PROGRAM MAIN
VAR
	
axis: AXIS_REF;
power: MC_POWER();

limNeg AT %I* :BOOL;
limPos AT %I*:BOOL;


EPSlimNeg AT %I* :BOOL;
EPSlimPos AT %I*:BOOL;

Ref:BOOL:=FALSE;
END_VAR

power(
	Axis:= axis, 
	Enable:= , 
	Enable_Positive:= limPos AND EPSlimPos, 
	Enable_Negative:= limNeg AND EPSlimNeg, 
	Override:= , 
	BufferMode:= , 
	Options:= , 
	Status=> , 
	Busy=> , 
	Active=> , 
	Error=> , 
	ErrorID=> );

END_PROGRAM

(* stored: Version 1.1.0.1, ProductVersion 3.1.4022.18
   POU MAIN: Id {cc9bc050-821b-46d6-9e4b-bb7db941681d}, SpecialFunc None *)
